(* Logix 5000 project; controller PBS_Perfusion vendor 1 type 14 code 217 rev 32.14; software revision 32.03; part 12 of 27 *)
(* tags used below, declared in another part *)
   Inp_OvrdCmd : DINT;   // Override Device Command: 0=None, 1=St.0, 2=St.1, 3=St.2, 4=St.3
   Cfg_NumStates : DINT;   // Number of device states (2..4)
   Cfg_OutSt0Write : SINT;   // Bit=1: write output in state 0, Bit=0: leave in last state
   Cfg_OutSt0State : SINT;   // (if written) Bit=1: output set in State 0, Bit=0: output cleared
   Cfg_OutSt1Write : SINT;   // Bit=1: write output in state 1, Bit=0: leave in last state
   Cfg_OutSt1State : SINT;   // (if written) Bit=1: output set in State 1, Bit=0: output cleared
   Cfg_OutSt2Write : SINT;   // Bit=1: write output in state 2, Bit=0: leave in last state
   Cfg_OutSt2State : SINT;   // (if written) Bit=1: output set in State 2, Bit=0: output cleared
   Cfg_OutSt3Write : SINT;   // Bit=1: write output in state 3, Bit=0: leave in last state
   Cfg_OutSt3State : SINT;   // (if written) Bit=1: output set in State 3, Bit=0: output cleared
   Cfg_FdbkSt0Check : SINT;   // Bit=1: Check Feedback in state 0, Bit=0: don't care
   Cfg_FdbkSt1Check : SINT;   // Bit=1: Check Feedback in state 1, Bit=0: don't care
   Cfg_FdbkSt2Check : SINT;   // Bit=1: Check Feedback in state 2, Bit=0: don't care
   Cfg_FdbkSt3Check : SINT;   // Bit=1: Check Feedback in state 3, Bit=0: don't care
   Cfg_OperSt0Prio : BOOL;   // 1=OCmd_St0 any time, 0=OCmd_St0 only when Oper selected
   Cfg_OCmdResets : BOOL;   // 1=New device OCmd resets shed latches and cleared alarms, 0=OCmdReset req'd.
   PSet_Owner : DINT;   // Program Owner Request ID (non-zero) or Release (zero)
   PCmd_St0 : BOOL;   // Program Command to set device to State 0
   PCmd_St1 : BOOL;   // Program Command to set device to State 1
   PCmd_St2 : BOOL;   // Program Command to set device to State 2
   PCmd_St3 : BOOL;   // Program Command to set device to State 3
   XCmd_St0 : BOOL;   // External Command to set device to State 0
   XCmd_St1 : BOOL;   // External Command to set device to State 1
   XCmd_St2 : BOOL;   // External Command to set device to State 2
   XCmd_St3 : BOOL;   // External Command to set device to State 3
   Out_A : BOOL;   // Output A to Device
   Out_B : BOOL;   // Output B to Device
   Out_C : BOOL;   // Output C to Device
   Out_D : BOOL;   // Output D to Device
   Out_Horn : BOOL;   // 1=Sound audible prior to commanded energize/ state change
   Val_Cmd : DINT;   // Device Command 0=None, 1=State 0, 2=State 1, 3=State 2, 4=State 3
   Val_Owner : DINT;   // Current Object Owner ID (0=not owned)
   Sts_St0 : BOOL;   // 1=Device commanded to and confirmed in State 0
   Sts_St1 : BOOL;   // 1=Device commanded to and confirmed in State 1
   Sts_St2 : BOOL;   // 1=Device commanded to and confirmed in State 2
   Sts_St3 : BOOL;   // 1=Device commanded to and confirmed in State 3
   Sts_Moving : BOOL;   // 1=Device not yet confirmed in commended state
   Sts_Horn : BOOL;   // 1=Sound audible prior to commanded energize/ state change
   Sts_NotRdy : BOOL;   // 1=Device Not Ready, see detail bits for reason
   Nrdy_CfgErr : BOOL;   // 1=Device Not Ready: Configuration Error
   Nrdy_EqpFault : BOOL;   // 1=Device Not Ready: External Equipment Fault (Fault or Shed Requires Reset)
   Nrdy_Fail : BOOL;   // 1=Device Not Ready: Device Failure (Shed Requires Reset)
   Nrdy_IOFault : BOOL;   // 1=Device Not Ready: I/O Fault (Shed Requires Reset)
   Nrdy_PrioSt0 : BOOL;   // 1=Device Not Ready: Oper/Ext Priority State 0 Command Requires Reset
   Nrdy_Perm : BOOL;   // 1=Device Not Ready: Permissive Not OK
   Sts_OoS : ALIAS FOR CmdSrc.Sts_OoS;
   Sts_Maint : ALIAS FOR CmdSrc.Sts_Maint;
   Sts_Oper : ALIAS FOR CmdSrc.Sts_Oper;
   Sts_DeviceFault : ALIAS FOR DeviceFault.Inp;   // 1=Device Fault (from Inp_DeviceFault)
   P_D4SD : BOOL;   // Unique Parameter Name for auto - discovery
   Wrk_OutDPulseT : TIMER;   // Output D Pulse Timer
   Wrk_OutCPulseT : TIMER;   // Output C Pulse Timer
   Wrk_OutBPulseT : TIMER;   // Output B Pulse Timer
   Wrk_OutAPulseT : TIMER;   // Output A Pulse Timer
   Wrk_ActState : DINT;   // Actual State (enum)
   Fail : P_Alarm;   // Device Fail to reach commanded position
   DeviceFault : P_Alarm;   // Device Fault from device via input
   CmdSrc : P_CmdSrc;   // Control / Command Source Selection
   IntlkTrip : P_Alarm;   // Interlock Trip Alarm
   Wrk_Out : SINT;   // Outputs (buffered) as a SINT for byte-wise operations
   Wrk_PermOK3 : BOOL;   // 1=Permissives are OK to go to state 3
   Wrk_PermOK2 : BOOL;   // 1=Permissives are OK to go to state 2
   Wrk_PermOK1 : BOOL;   // 1=Permissives are OK to go to state 1
   Wrk_PermOK0 : BOOL;   // 1=Permissives are OK to go to state 0
   Wrk_TgtState : DINT;   // Target device state as a number (0, 1, 2 or 3)
   Wrk_NewCmd : BOOL;   // 1=A state command has been received (even for same state)
   Wrk_PrevTgt : DINT;   // Previous Target State (last scan)
   Wrk_NotRdy : BOOL;   // Device Not Ready conditions excluding shed latches
   ORdy_St3 : BOOL;   // 1=Ready for OCmd_St3, enable HMI button
   ORdy_St2 : BOOL;   // 1=Ready for OCmd_St2, enable HMI button
   ORdy_St1 : BOOL;   // 1=Ready for OCmd_St1, enable HMI button
   ORdy_St0 : BOOL;   // 1=Ready for OCmd_St0, enable HMI button
   MRdy_Check : BOOL;   // 1=Ready for MCmd_Check, enable HMI button
   MRdy_Bypass : BOOL;   // 1=Ready for MCmd_Bypass, enable HMI button
   OCmd_St3 : BOOL;   // Operator Command to set device to State 3
   OCmd_St2 : BOOL;   // Operator Command to set device to State 2
   OCmd_St1 : BOOL;   // Operator Command to set device to State 1
   OCmd_St0 : BOOL;   // Operator Command to set device to State 0
   MCmd_Check : BOOL;   // Maintenance Command to Check Interlocks and Permissives
   MCmd_Bypass : BOOL;   // Maintenance Command to Bypass Interlocks and Permissives
   Wrk_StartHorn : BOOL;   // 1=Sound audible prior to commanded energize/ state change
   REAL : DINT;
(* P_D4SD, continued *)

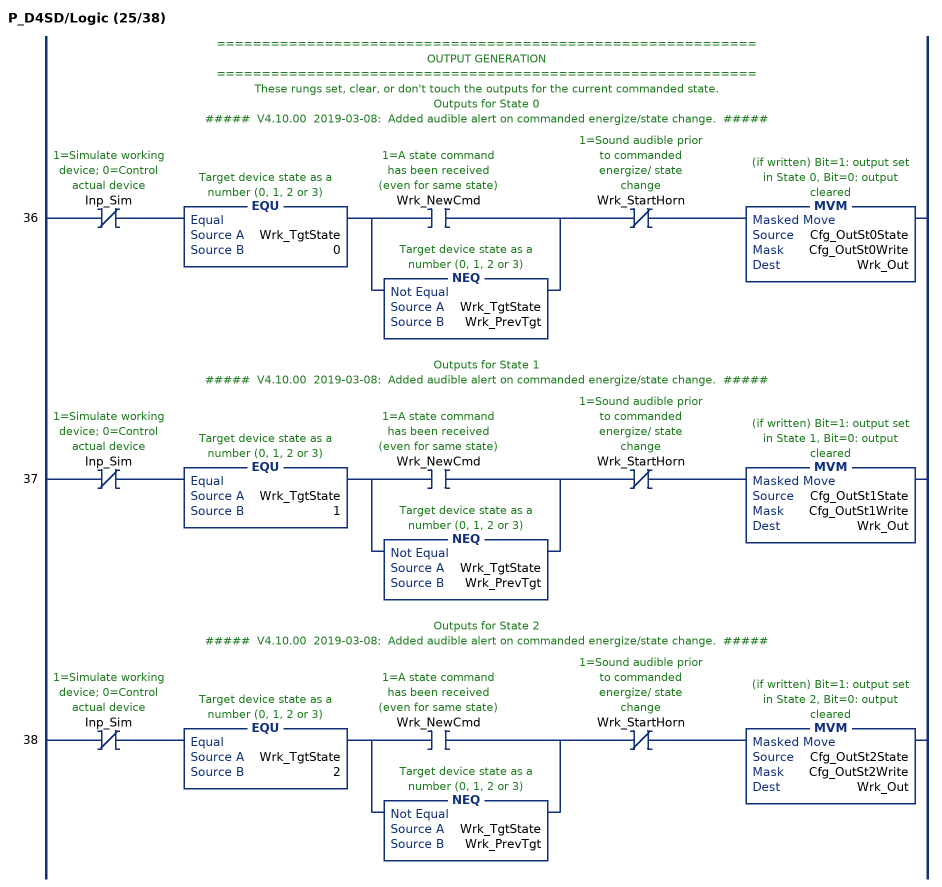
   // ============================================================
   // OUTPUT GENERATION
   // ============================================================
   // These rungs set, clear, or don't touch the outputs for the current commanded state.
   // Outputs for State 0
   // #####  V4.10.00  2019-03-08:  Added audible alert on commanded energize/state change.  #####
   36: XIO(Inp_Sim)EQU(Wrk_TgtState,0)[XIC(Wrk_NewCmd) ,NEQ(Wrk_TgtState,Wrk_PrevTgt) ]XIO(Wrk_StartHorn)MVM(Cfg_OutSt0State,Cfg_OutSt0Write,Wrk_Out);
   // Outputs for State 1
   // #####  V4.10.00  2019-03-08:  Added audible alert on commanded energize/state change.  #####
   37: XIO(Inp_Sim)EQU(Wrk_TgtState,1)[XIC(Wrk_NewCmd) ,NEQ(Wrk_TgtState,Wrk_PrevTgt) ]XIO(Wrk_StartHorn)MVM(Cfg_OutSt1State,Cfg_OutSt1Write,Wrk_Out);
   // Outputs for State 2
   // #####  V4.10.00  2019-03-08:  Added audible alert on commanded energize/state change.  #####
   38: XIO(Inp_Sim)EQU(Wrk_TgtState,2)[XIC(Wrk_NewCmd) ,NEQ(Wrk_TgtState,Wrk_PrevTgt) ]XIO(Wrk_StartHorn)MVM(Cfg_OutSt2State,Cfg_OutSt2Write,Wrk_Out);
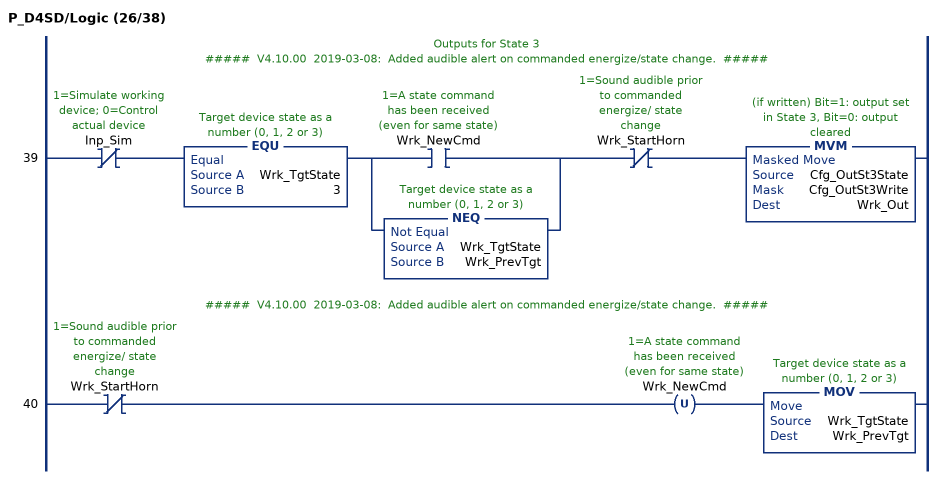
   // Outputs for State 3
   // #####  V4.10.00  2019-03-08:  Added audible alert on commanded energize/state change.  #####
   39: XIO(Inp_Sim)EQU(Wrk_TgtState,3)[XIC(Wrk_NewCmd) ,NEQ(Wrk_TgtState,Wrk_PrevTgt) ]XIO(Wrk_StartHorn)MVM(Cfg_OutSt3State,Cfg_OutSt3Write,Wrk_Out);
   // #####  V4.10.00  2019-03-08:  Added audible alert on commanded energize/state change.  #####
   40: XIO(Wrk_StartHorn)OTU(Wrk_NewCmd)MOV(Wrk_TgtState,Wrk_PrevTgt);
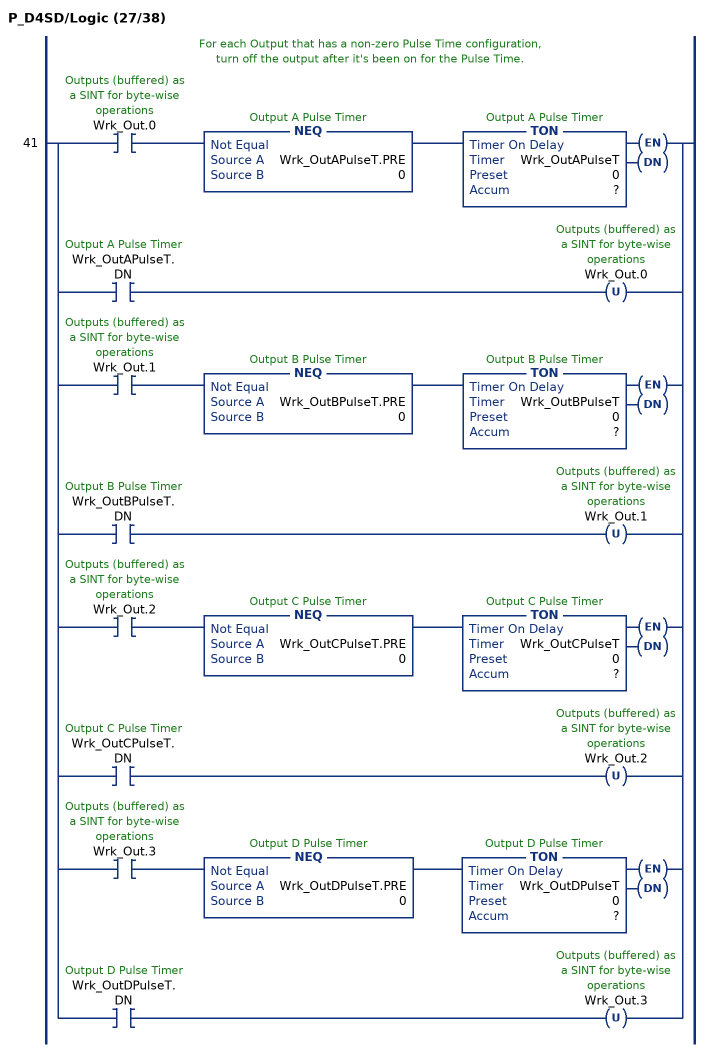
   // For each Output that has a non-zero Pulse Time configuration,
   // turn off the output after it's been on for the Pulse Time.
   41: [XIC(Wrk_Out.0) NEQ(Wrk_OutAPulseT.PRE,0) TON(Wrk_OutAPulseT,?,?) ,XIC(Wrk_OutAPulseT.DN) OTU(Wrk_Out.0) ,XIC(Wrk_Out.1) NEQ(Wrk_OutBPulseT.PRE,0) TON(Wrk_OutBPulseT,?,?) ,XIC(Wrk_OutBPulseT.DN) OTU(Wrk_Out.1) ,XIC(Wrk_Out.2) NEQ(Wrk_OutCPulseT.PRE,0) TON(Wrk_OutCPulseT,?,?) ,XIC(Wrk_OutCPulseT.DN) OTU(Wrk_Out.2) ,XIC(Wrk_Out.3) NEQ(Wrk_OutDPulseT.PRE,0) TON(Wrk_OutDPulseT,?,?) ,XIC(Wrk_OutDPulseT.DN) OTU(Wrk_Out.3) ];
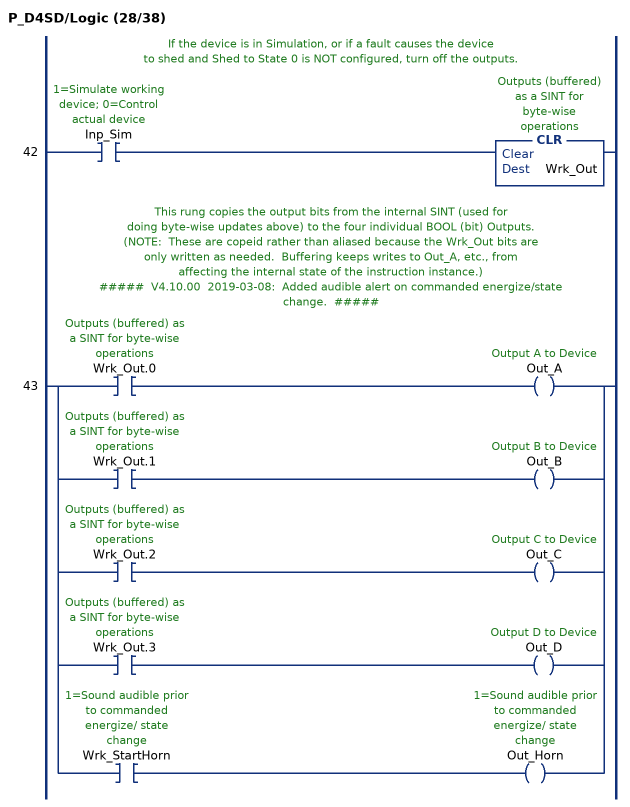
   // If the device is in Simulation, or if a fault causes the device
   // to shed and Shed to State 0 is NOT configured, turn off the outputs.
   42: XIC(Inp_Sim)CLR(Wrk_Out);
   // This rung copies the output bits from the internal SINT (used for
   // doing byte-wise updates above) to the four individual BOOL (bit) Outputs.
   // (NOTE:  These are copeid rather than aliased because the Wrk_Out bits are
   // only written as needed.  Buffering keeps writes to Out_A, etc., from
   // affecting the internal state of the instruction instance.)
   // #####  V4.10.00  2019-03-08:  Added audible alert on commanded energize/state change.  #####
   43: [XIC(Wrk_Out.0) OTE(Out_A) ,XIC(Wrk_Out.1) OTE(Out_B) ,XIC(Wrk_Out.2) OTE(Out_C) ,XIC(Wrk_Out.3) OTE(Out_D) ,XIC(Wrk_StartHorn) OTE(Out_Horn) ];
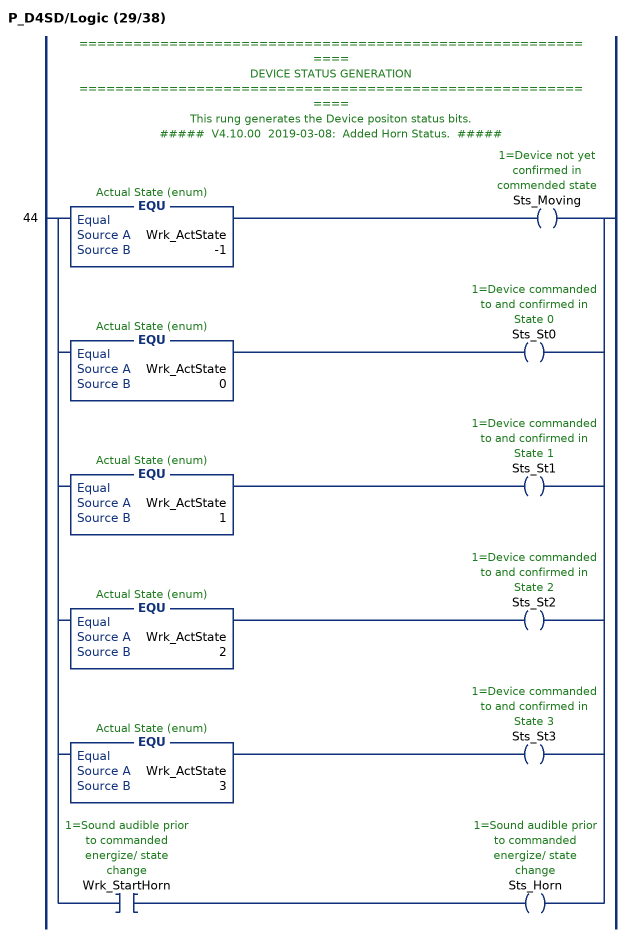
   // ============================================================
   // DEVICE STATUS GENERATION
   // ============================================================
   // This rung generates the Device positon status bits.
   // #####  V4.10.00  2019-03-08:  Added Horn Status.  #####
   44: [EQU(Wrk_ActState,-1) OTE(Sts_Moving) ,EQU(Wrk_ActState,0) OTE(Sts_St0) ,EQU(Wrk_ActState,1) OTE(Sts_St1) ,EQU(Wrk_ActState,2) OTE(Sts_St2) ,EQU(Wrk_ActState,3) OTE(Sts_St3) ,XIC(Wrk_StartHorn) OTE(Sts_Horn) ];
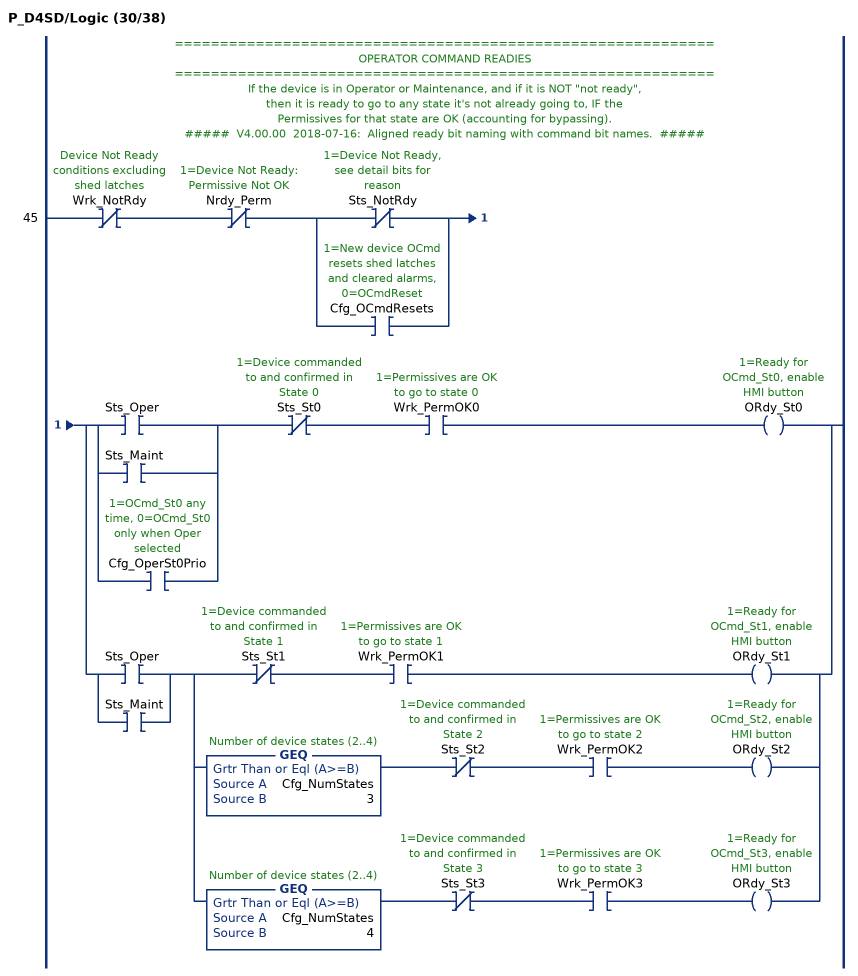
   // ============================================================
   // OPERATOR COMMAND READIES
   // ============================================================
   // If the device is in Operator or Maintenance, and if it is NOT "not ready",
   // then it is ready to go to any state it's not already going to, IF the
   // Permissives for that state are OK (accounting for bypassing).
   // #####  V4.00.00  2018-07-16:  Aligned ready bit naming with command bit names.  #####
   45: XIO(Wrk_NotRdy)XIO(Nrdy_Perm)[XIO(Sts_NotRdy) ,XIC(Cfg_OCmdResets) ][[XIC(Sts_Oper) ,XIC(Sts_Maint) ,XIC(Cfg_OperSt0Prio) ] XIO(Sts_St0) XIC(Wrk_PermOK0) OTE(ORdy_St0) ,[XIC(Sts_Oper) ,XIC(Sts_Maint) ] [XIO(Sts_St1) XIC(Wrk_PermOK1) OTE(ORdy_St1) ,GEQ(Cfg_NumStates,3) XIO(Sts_St2) XIC(Wrk_PermOK2) OTE(ORdy_St2) ,GEQ(Cfg_NumStates,4) XIO(Sts_St3) XIC(Wrk_PermOK3) OTE(ORdy_St3) ] ];
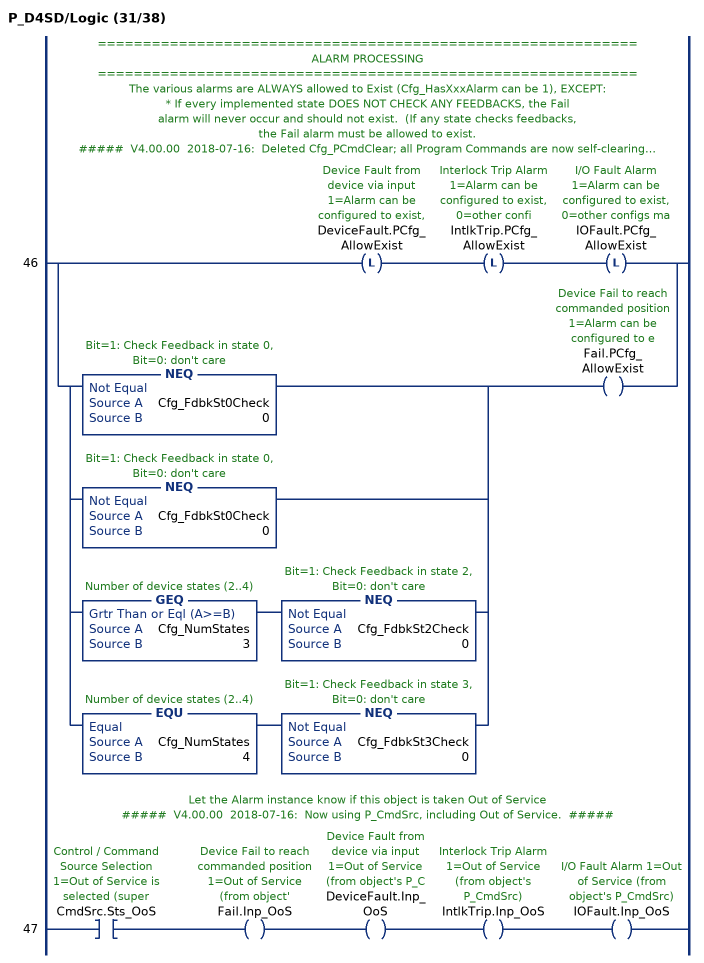
   // ============================================================
   // ALARM PROCESSING
   // ============================================================
   // The various alarms are ALWAYS allowed to Exist (Cfg_HasXxxAlarm can be 1), EXCEPT:
   // * If every implemented state DOES NOT CHECK ANY FEEDBACKS, the Fail
   // alarm will never occur and should not exist.  (If any state checks feedbacks,
   // the Fail alarm must be allowed to exist.
   // #####  V4.00.00  2018-07-16:  Deleted Cfg_PCmdClear; all Program Commands are now self-clearing.  #####
   46: [OTL(DeviceFault.PCfg_AllowExist) OTL(IntlkTrip.PCfg_AllowExist) OTL(IOFault.PCfg_AllowExist) ,[NEQ(Cfg_FdbkSt0Check,0) ,NEQ(Cfg_FdbkSt0Check,0) ,GEQ(Cfg_NumStates,3) NEQ(Cfg_FdbkSt2Check,0) ,EQU(Cfg_NumStates,4) NEQ(Cfg_FdbkSt3Check,0) ] OTE(Fail.PCfg_AllowExist) ];
   // Let the Alarm instance know if this object is taken Out of Service
   // #####  V4.00.00  2018-07-16:  Now using P_CmdSrc, including Out of Service.  #####
   47: XIC(CmdSrc.Sts_OoS)OTE(Fail.Inp_OoS)OTE(DeviceFault.Inp_OoS)OTE(IntlkTrip.Inp_OoS)OTE(IOFault.Inp_OoS);
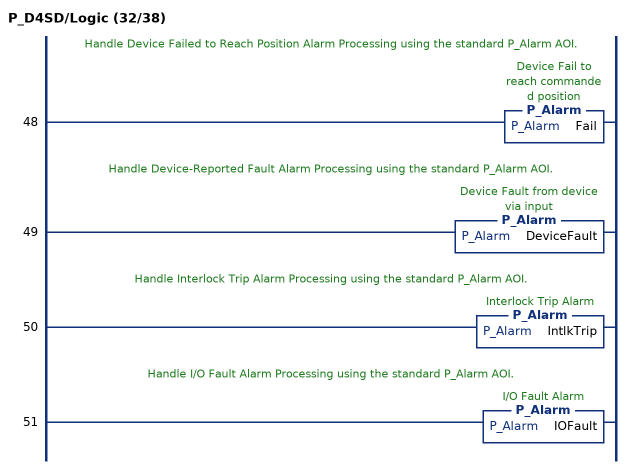
   // Handle Device Failed to Reach Position Alarm Processing using the standard P_Alarm AOI.
   48: P_Alarm(Fail);
   // Handle Device-Reported Fault Alarm Processing using the standard P_Alarm AOI.
   49: P_Alarm(DeviceFault);
   // Handle Interlock Trip Alarm Processing using the standard P_Alarm AOI.
   50: P_Alarm(IntlkTrip);
   // Handle I/O Fault Alarm Processing using the standard P_Alarm AOI.
   51: P_Alarm(IOFault);
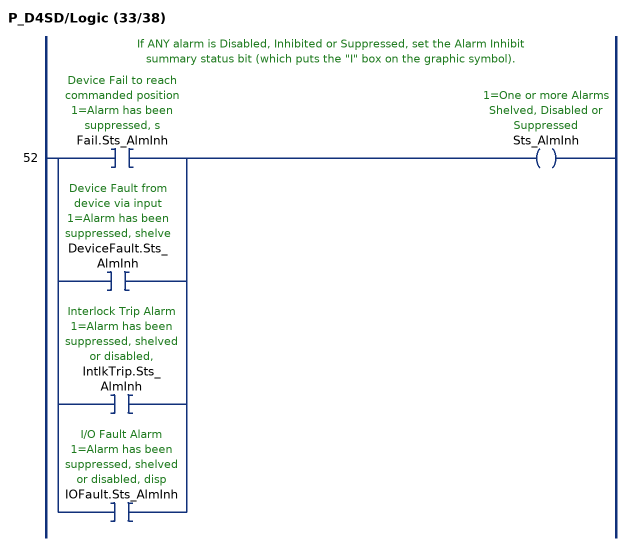
   // If ANY alarm is Disabled, Inhibited or Suppressed, set the Alarm Inhibit
   // summary status bit (which puts the "I" box on the graphic symbol).
   52: [XIC(Fail.Sts_AlmInh) ,XIC(DeviceFault.Sts_AlmInh) ,XIC(IntlkTrip.Sts_AlmInh) ,XIC(IOFault.Sts_AlmInh) ]OTE(Sts_AlmInh);
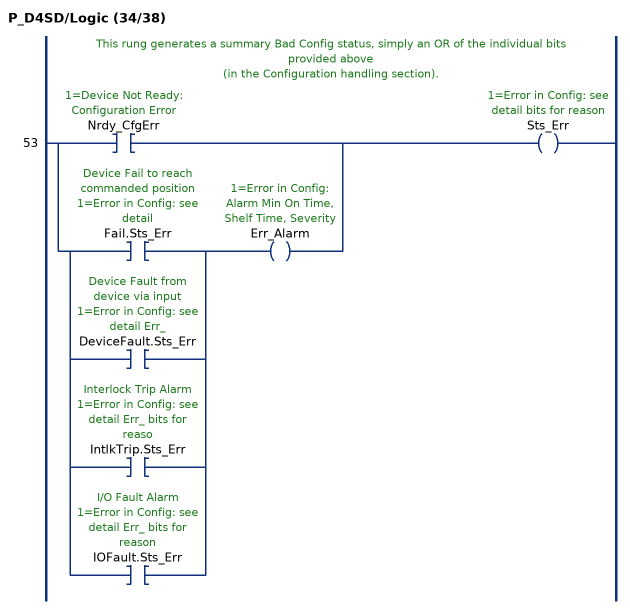
   // This rung generates a summary Bad Config status, simply an OR of the individual bits provided above
   // (in the Configuration handling section).
   53: [XIC(Nrdy_CfgErr) ,[XIC(Fail.Sts_Err) ,XIC(DeviceFault.Sts_Err) ,XIC(IntlkTrip.Sts_Err) ,XIC(IOFault.Sts_Err) ] OTE(Err_Alarm) ]OTE(Sts_Err);
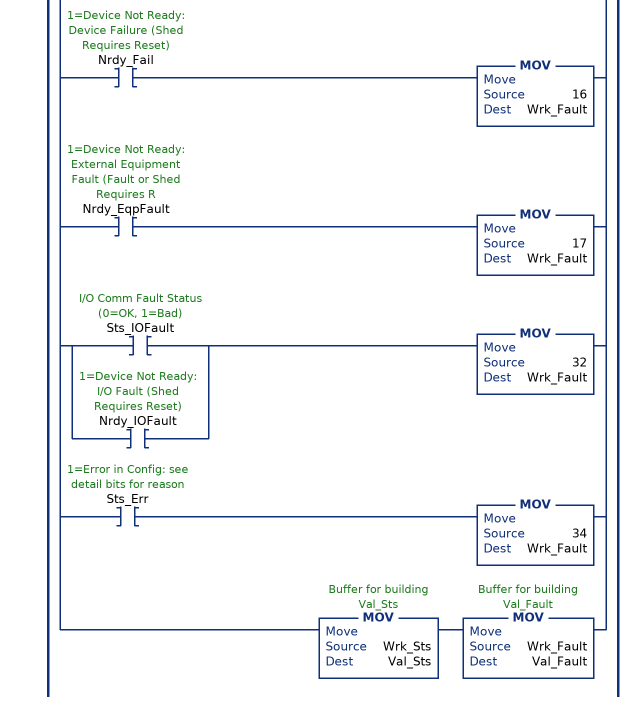
   // This rung generates the enumerated Device Status:
   // 0 = Powerup / Unknown
   // 1=Confirmed in State 0
   // 2 = Confirmed in State 1
   // 3 = Confirmed in State 2
   // 4 = Confirmed in State 3
   // 5 = Moving to new target State
   // 10 = Horn
   // And this rung generates the enumerated Device Fault Status:
   // 0 = none
   // 16 = Failed to reach commanded position
   // 17 = Device Fail (from input)
   // 32 = I/O Fault
   // 34 = Config Error
   // #####  V4.00.00  2018-07-16:  Disable/Enable replaced by P_CmdSrc Out of Service (OoS).  #####
   // #####  V4.10.00  2019-03-08:  Added Horn Status.  #####
   54: [CLR(Wrk_Sts) CLR(Wrk_Fault) ,XIC(Sts_St0) MOV(1,Wrk_Sts) ,XIC(Sts_St1) MOV(2,Wrk_Sts) ,XIC(Sts_St2) MOV(3,Wrk_Sts) ,XIC(Sts_St3) MOV(4,Wrk_Sts) ,XIC(Sts_Moving) MOV(9,Wrk_Sts) ,XIC(Sts_Horn) MOV(10,Wrk_Sts) ,XIC(Nrdy_Fail) MOV(16,Wrk_Fault) ,XIC(Nrdy_EqpFault) MOV(17,Wrk_Fault) ,[XIC(Sts_IOFault) ,XIC(Nrdy_IOFault) ] MOV(32,Wrk_Fault) ,XIC(Sts_Err) MOV(34,Wrk_Fault) ,MOV(Wrk_Sts,Val_Sts) MOV(Wrk_Fault,Val_Fault) ];
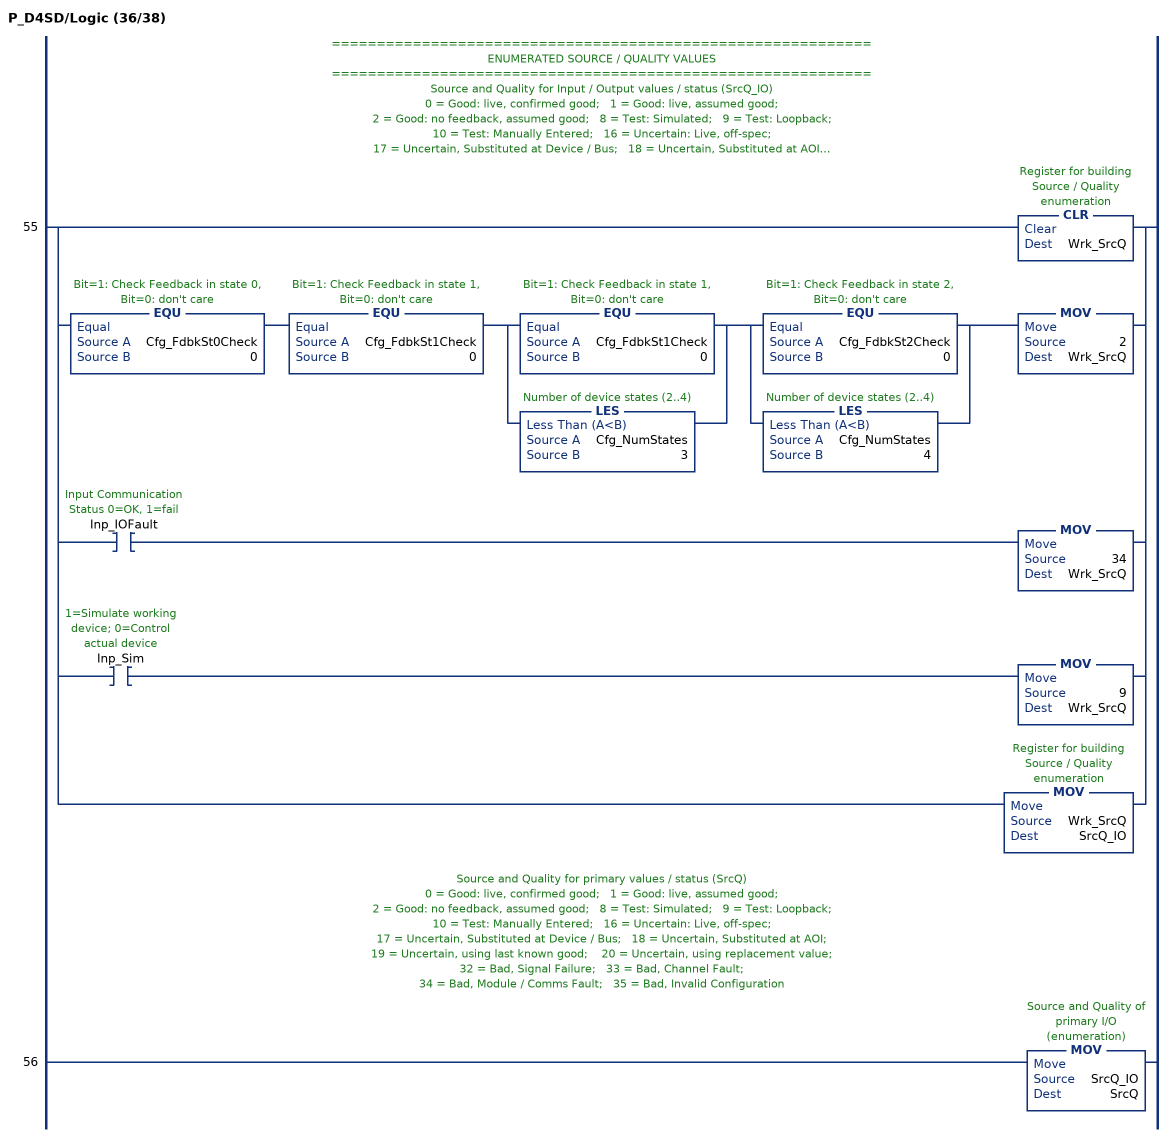
   // ============================================================
   // ENUMERATED SOURCE / QUALITY VALUES
   // ============================================================
   // Source and Quality for Input / Output values / status (SrcQ_IO)
   // 0 = Good: live, confirmed good;   1 = Good: live, assumed good;
   // 2 = Good: no feedback, assumed good;   8 = Test: Simulated;   9 = Test: Loopback;
   // 10 = Test: Manually Entered;   16 = Uncertain: Live, off-spec;
   // 17 = Uncertain, Substituted at Device / Bus;   18 = Uncertain, Substituted at AOI;
   // 19 = Uncertain, using last known good;    20 = Uncertain, using replacement value;
   // 32 = Bad, Signal Failure;   33 = Bad, Channel Fault;
   // 34 = Bad, Module / Comms Fault;   35 = Bad, Invalid Configuration.
   55: [CLR(Wrk_SrcQ) ,EQU(Cfg_FdbkSt0Check,0) EQU(Cfg_FdbkSt1Check,0) [EQU(Cfg_FdbkSt1Check,0) ,LES(Cfg_NumStates,3) ] [EQU(Cfg_FdbkSt2Check,0) ,LES(Cfg_NumStates,4) ] MOV(2,Wrk_SrcQ) ,XIC(Inp_IOFault) MOV(34,Wrk_SrcQ) ,XIC(Inp_Sim) MOV(9,Wrk_SrcQ) ,MOV(Wrk_SrcQ,SrcQ_IO) ];
   // Source and Quality for primary values / status (SrcQ)
   // 0 = Good: live, confirmed good;   1 = Good: live, assumed good;
   // 2 = Good: no feedback, assumed good;   8 = Test: Simulated;   9 = Test: Loopback;
   // 10 = Test: Manually Entered;   16 = Uncertain: Live, off-spec;
   // 17 = Uncertain, Substituted at Device / Bus;   18 = Uncertain, Substituted at AOI;
   // 19 = Uncertain, using last known good;    20 = Uncertain, using replacement value;
   // 32 = Bad, Signal Failure;   33 = Bad, Channel Fault;
   // 34 = Bad, Module / Comms Fault;   35 = Bad, Invalid Configuration
   56: MOV(SrcQ_IO,SrcQ);
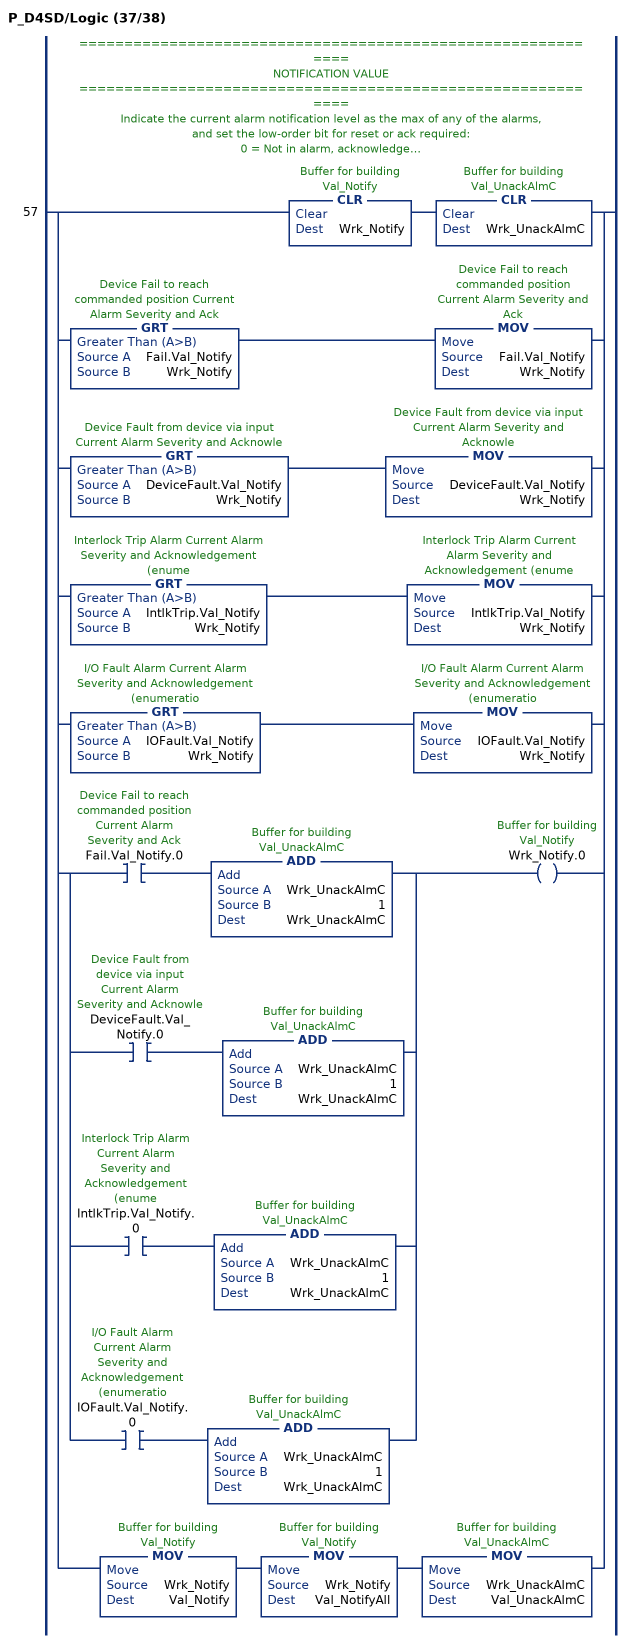
   // ============================================================
   // NOTIFICATION VALUE
   // ============================================================
   // Indicate the current alarm notification level as the max of any of the alarms,
   // and set the low-order bit for reset or ack required:
   // 0 = Not in alarm, acknowledged
   // 1 = Not in alarm, unacknowledged or reset required
   // 2 = Low severity alarm, acknowledged
   // 3 = Low severity alarm, unacknowledged
   // 4 = Medium severity alarm, acknowledged
   // 5 = Medium severity alarm, unacknowledged
   // 6 = High severity alarm, acknowledged
   // 7 = High severity alarm, unacknowledged
   // 8 = Urgent severity alarm, acknowledged
   // 9 = Urgent severity alarm, unacknowledged
   // #####  V4.00.00  2018-07-16:  Added Val_NotifyAll and Val_UnackAlmC to roll up alarm  #####
   // #####  priority / ack status and unack. alarm count.  #####
   57: [CLR(Wrk_Notify) CLR(Wrk_UnackAlmC) ,GRT(Fail.Val_Notify,Wrk_Notify) MOV(Fail.Val_Notify,Wrk_Notify) ,GRT(DeviceFault.Val_Notify,Wrk_Notify) MOV(DeviceFault.Val_Notify,Wrk_Notify) ,GRT(IntlkTrip.Val_Notify,Wrk_Notify) MOV(IntlkTrip.Val_Notify,Wrk_Notify) ,GRT(IOFault.Val_Notify,Wrk_Notify) MOV(IOFault.Val_Notify,Wrk_Notify) ,[XIC(Fail.Val_Notify.0) ADD(Wrk_UnackAlmC,1,Wrk_UnackAlmC) ,XIC(DeviceFault.Val_Notify.0) ADD(Wrk_UnackAlmC,1,Wrk_UnackAlmC) ,XIC(IntlkTrip.Val_Notify.0) ADD(Wrk_UnackAlmC,1,Wrk_UnackAlmC) ,XIC(IOFault.Val_Notify.0) ADD(Wrk_UnackAlmC,1,Wrk_UnackAlmC) ] OTE(Wrk_Notify.0) ,MOV(Wrk_Notify,Val_Notify) MOV(Wrk_Notify,Val_NotifyAll) MOV(Wrk_UnackAlmC,Val_UnackAlmC) ];
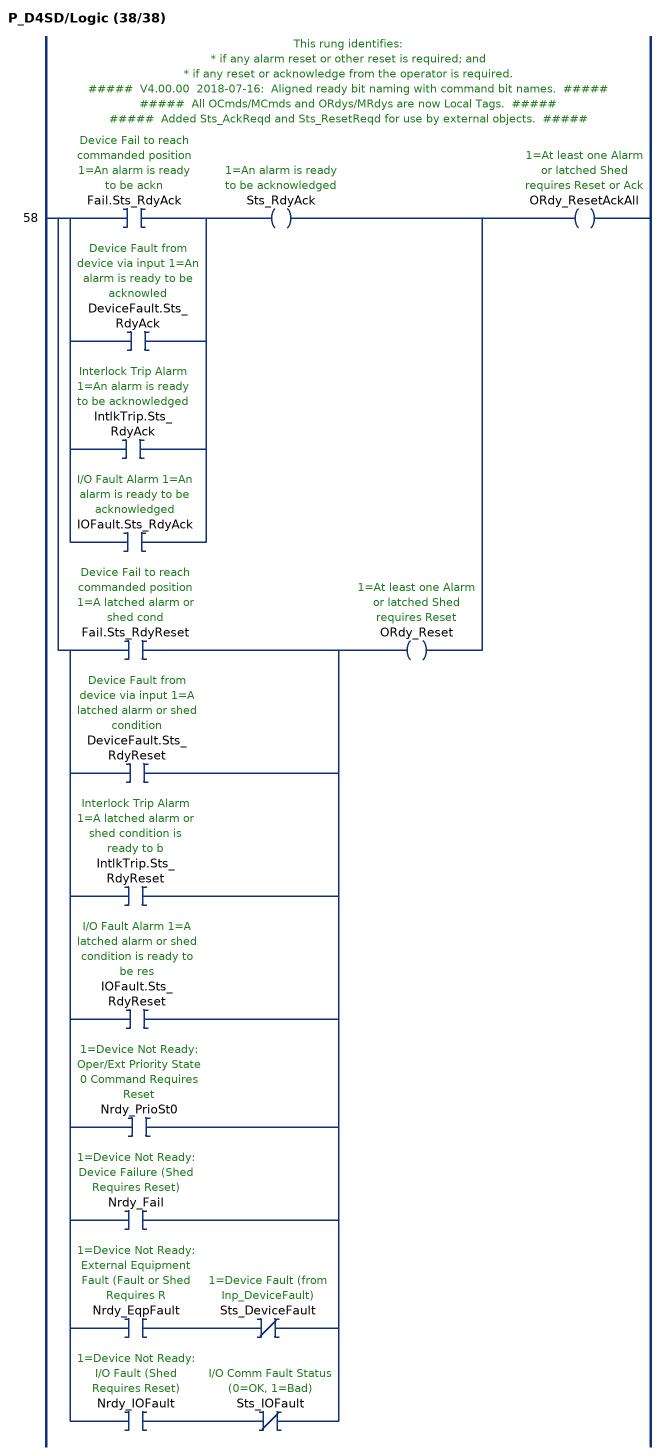
   // This rung identifies:
   // * if any alarm reset or other reset is required; and
   // * if any reset or acknowledge from the operator is required.
   // #####  V4.00.00  2018-07-16:  Aligned ready bit naming with command bit names.  #####
   // #####  All OCmds/MCmds and ORdys/MRdys are now Local Tags.  #####
   // #####  Added Sts_AckReqd and Sts_ResetReqd for use by external objects.  #####
   58: [[XIC(Fail.Sts_RdyAck) ,XIC(DeviceFault.Sts_RdyAck) ,XIC(IntlkTrip.Sts_RdyAck) ,XIC(IOFault.Sts_RdyAck) ] OTE(Sts_RdyAck) ,[XIC(Fail.Sts_RdyReset) ,XIC(DeviceFault.Sts_RdyReset) ,XIC(IntlkTrip.Sts_RdyReset) ,XIC(IOFault.Sts_RdyReset) ,XIC(Nrdy_PrioSt0) ,XIC(Nrdy_Fail) ,XIC(Nrdy_EqpFault) XIO(Sts_DeviceFault) ,XIC(Nrdy_IOFault) XIO(Sts_IOFault) ] OTE(ORdy_Reset) ]OTE(ORdy_ResetAckAll);
END_ROUTINE

ROUTINE Prescan   (* ladder *)
// Clear Ownership, clear "lurking" Commands
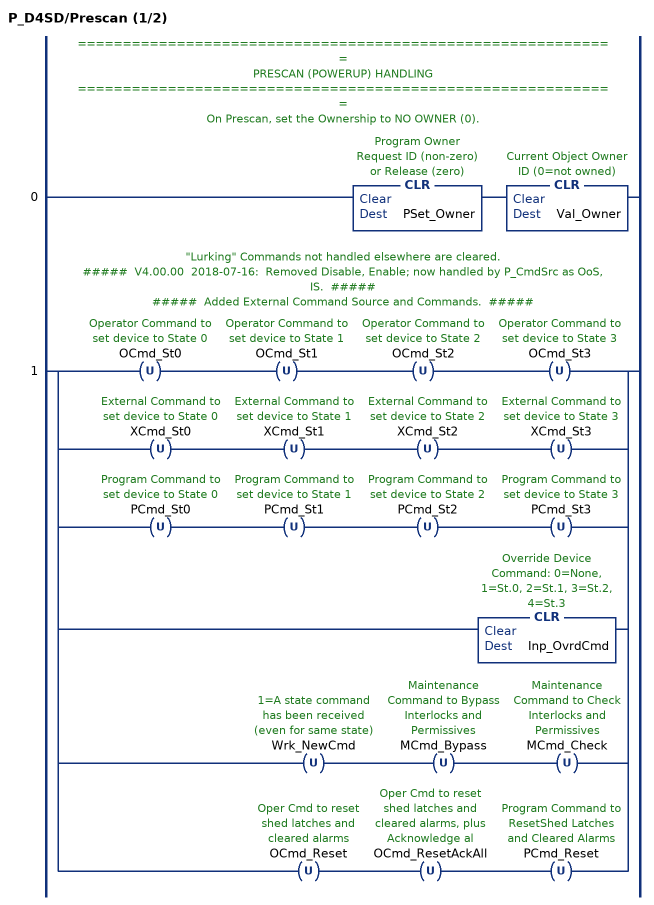
   // ============================================================
   // PRESCAN (POWERUP) HANDLING
   // ============================================================
   // On Prescan, set the Ownership to NO OWNER (0).
   0: CLR(PSet_Owner)CLR(Val_Owner);
   // "Lurking" Commands not handled elsewhere are cleared.
   // #####  V4.00.00  2018-07-16:  Removed Disable, Enable; now handled by P_CmdSrc as OoS, IS.  #####
   // #####  Added External Command Source and Commands.  #####
   1: [OTU(OCmd_St0) OTU(OCmd_St1) OTU(OCmd_St2) OTU(OCmd_St3) ,OTU(XCmd_St0) OTU(XCmd_St1) OTU(XCmd_St2) OTU(XCmd_St3) ,OTU(PCmd_St0) OTU(PCmd_St1) OTU(PCmd_St2) OTU(PCmd_St3) ,CLR(Inp_OvrdCmd) ,OTU(Wrk_NewCmd) OTU(MCmd_Bypass) OTU(MCmd_Check) ,OTU(OCmd_Reset) OTU(OCmd_ResetAckAll) OTU(PCmd_Reset) ];
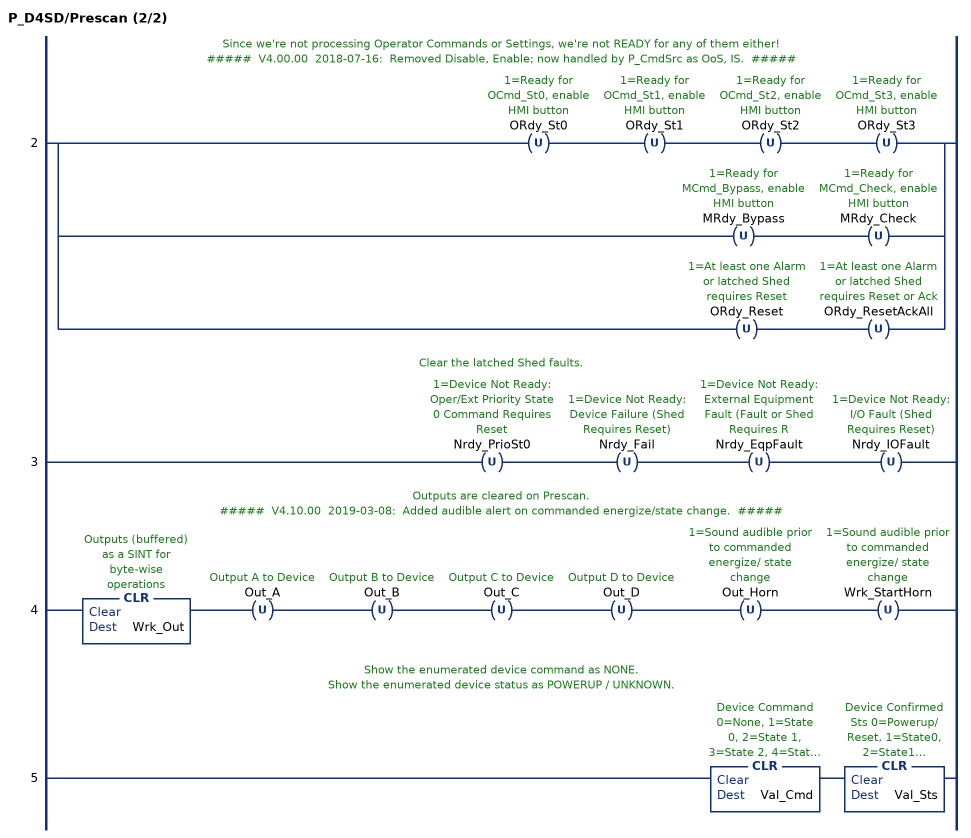
   // Since we're not processing Operator Commands or Settings, we're not READY for any of them either!
   // #####  V4.00.00  2018-07-16:  Removed Disable, Enable; now handled by P_CmdSrc as OoS, IS.  #####
   2: [OTU(ORdy_St0) OTU(ORdy_St1) OTU(ORdy_St2) OTU(ORdy_St3) ,OTU(MRdy_Bypass) OTU(MRdy_Check) ,OTU(ORdy_Reset) OTU(ORdy_ResetAckAll) ];
   // Clear the latched Shed faults.
   3: OTU(Nrdy_PrioSt0)OTU(Nrdy_Fail)OTU(Nrdy_EqpFault)OTU(Nrdy_IOFault);
   // Outputs are cleared on Prescan.
   // #####  V4.10.00  2019-03-08:  Added audible alert on commanded energize/state change.  #####
   4: CLR(Wrk_Out)OTU(Out_A)OTU(Out_B)OTU(Out_C)OTU(Out_D)OTU(Out_Horn)OTU(Wrk_StartHorn);
   // Show the enumerated device command as NONE.
   // Show the enumerated device status as POWERUP / UNKNOWN.
   5: CLR(Val_Cmd)CLR(Val_Sts);
END_ROUTINE
END_ADD_ON_INSTRUCTION

ADD_ON_INSTRUCTION P_DIn   (* revision 4.10 .00 Release, vendor Rockwell Automation, ExecutePrescan, ExecuteEnableInFalse *)
// Discrete Input
// Revision note:
// See Instruction Help for a summary of changes, and see 4.10 Release Notes for details.
// Help:
// Copyright © Rockwell Automation, Inc.  All Rights Reserved.
// This instruction monitors a discrete (1 / 0) input and checks for alarm conditions.
// The Inp_Gate input must be set (=1, its default value) and the alarm enabled for
// the Target Disagree alarm to occur.  This alarm will not occur until the Inp_Gate
// input has been set for the Gate Delay (Cfg_GateDly) time.  The Gate is used to
// enable the alarm when some other condition is true; for example, a high vibration
// switch should only generate a Target Disagree alarm when the associated motor
// has been running long enough to stabilize.
// The Target Disagree alarm is generated when the Inp_PV (process variable)
// input is different from the Inp_Target (target) input.  The Target indicates the
// "normal" condition.  For example, a flow switch should indicate flow when a
// pump is running and should not indicate flow when a pump is stopped.  The
// pump run status is used as the Target input, and when the switch does not
// match the target (within the allotted time), the Target Disagree Alarm (e.g.,
// Flow Switch Failure) is generated.
// NOTE: the Inp_PV is inverted when the rung condition is false -- this allows the
// input to be a condition on the rung with P_DIn rather than mapped into Inp_PV.
// See P_DIn reference manual for details.
// This instruction includes a substitute PV capability for a manually-entered state.
// This may be useful when a sensor is out for repair or for simulation and testing.
// Alarms are provided by P_Alarm AOI instances.
// Target Disagree Status gating provided by a P_Gate AOI instance.
// SUMMARY OF CHANGES FROM PREVIOUS VERSION (4.00.00)
// See 4.10 Release Notes for details.
// * Added Cfg_HasMoreObj.
// SUMMARY OF CHANGES FROM PREVIOUS VERSION (3.5-01)
// See 4.00 Release Notes for details.
// * Changed Inf_ items to HMI_, and added Cfg_Area for security.
// * Added notify and unack count rollup for Channel object.
// * Added I/O Fault alarm.
// * Deleted Cfg_PCmdClear.  All Program Commands are now self-clearing.
// * Aligned ready bit naming with command bit names.
// * All OCmds/MCmds and ORdys/MRdys are now Local Tags.
// * Added Sts_RdyAck and Sts_RdyReset for use by external objects.
// * Changed delay time configuration items to REAL seconds.
VAR_INPUT
   Inp_PV : BOOL := 1; {visible}   // Input Signal (process variable) from Sensor
   Inp_IOFault : BOOL; {visible}   // Input Comm Status or Quality 1=Bad, 0=OK
   Inp_PVNotify : DINT;   // Related PV object alarm prio and ack status (enum)
   Inp_Target : BOOL := 1; {visible}   // Target State of Input (Disagree Status if not in Target State)
   Inp_Gate : ALIAS FOR TgtDisagreeGate.Inp_Gate; {visible}   // Gate Condition (=1 to enable Disagree Status)
   Inp_Sim : BOOL;   // 1=Use simulated PV (Set_SimPV); 0=Use Input (Inp_PV)
   Inp_Reset : BOOL;   // 1=Reset Alarm requiring reset
   Cfg_NoSubstPV : BOOL;   // 1=Disallow selection of Substitute PV
   Cfg_NormTextVis : BOOL := 1;   // 1=Display state text in "normal" state (= target), 0=hide (some HMI objects)
   Cfg_HasMoreObj : BOOL;   // 1=Tells HMI an object with more info is available
   Cfg_HasTgtDisagreeAlm : ALIAS FOR TgtDisagree.Cfg_Exists;   // 1=Target Disagree Alarm exists and will be checked
   Cfg_TgtDisagreeResetReqd : ALIAS FOR TgtDisagree.Cfg_ResetReqd;   // 1=Target Disagree Alarm is latched in, requires Reset Command to clear
   Cfg_TgtDisagreeAckReqd : ALIAS FOR TgtDisagree.Cfg_AckReqd;   // 1=Target Disagree Alarm must be acknowledged
   Cfg_HasIOFaultAlm : ALIAS FOR IOFault.Cfg_Exists;   // 1=Target Disagree Alarm exists and will be checked
   Cfg_IOFaultResetReqd : ALIAS FOR IOFault.Cfg_ResetReqd;   // 1=Target Disagree Alarm is latched in, requires Reset Command to clear
   Cfg_IOFaultAckReqd : ALIAS FOR IOFault.Cfg_AckReqd;   // 1=Target Disagree Alarm must be acknowledged
   Cfg_TgtDisagreeSeverity : ALIAS FOR TgtDisagree.Cfg_Severity;   // Target Disagree Alarm Severity: 1..250=Low, 251..500=Medium, 501..750=High, 751..1000=Urgent
   Cfg_IOFaultSeverity : ALIAS FOR IOFault.Cfg_Severity;   // Target Disagree Alarm Severity: 1..250=Low, 251..500=Medium, 501..750=High, 751..1000=Urgent
   Cfg_Debounce : REAL;   // Minimum time Input Sts must maintain state (sec)
   Cfg_GateDly : ALIAS FOR TgtDisagreeGate.Cfg_GateDly;   // Time Inp_Gate must be true before Disagree Status is checked (sec)
   Cfg_TgtDisagreeOnDly : ALIAS FOR TgtDisagreeGate.Cfg_OnDly;   // Minimum time for Input to disagree with Target to raise Status (sec)
   Cfg_TgtDisagreeOffDly : ALIAS FOR TgtDisagreeGate.Cfg_OffDly;   // Minimum time for Input to agree with Target to clear Status (sec)
   Set_SimPV : BOOL;   // PV used in Simulation (Inp_Sim=1)
   PCmd_Reset : BOOL;   // Program Command to Reset all latched Alarms
   PCmd_TgtDisagreeAck : ALIAS FOR TgtDisagree.PCmd_Ack;   // Program Command to Acknowledge the Target Disagree Alarm
   PCmd_TgtDisagreeSuppress : ALIAS FOR TgtDisagree.PCmd_Suppress;   // Program Command to Suppress the Target Disagree Alarm
   PCmd_TgtDisagreeUnsuppress : ALIAS FOR TgtDisagree.PCmd_Unsuppress;   // Program Command to Unsuppress the Target Disagree Alarm
   PCmd_TgtDisagreeUnshelve : ALIAS FOR TgtDisagree.PCmd_Unshelve;   // Program Command to Unshelve the Target Disagree Alarm
   PCmd_IOFaultAck : ALIAS FOR IOFault.PCmd_Ack;   // Program Command to Acknowledge the I/O Fault Alarm
   PCmd_IOFaultSuppress : ALIAS FOR IOFault.PCmd_Suppress;   // Program Command to Suppress the I/O Fault Alarm
   PCmd_IOFaultUnsuppress : ALIAS FOR IOFault.PCmd_Unsuppress;   // Program Command to Unsuppress the I/O Fault Alarm
   PCmd_IOFaultUnshelve : ALIAS FOR IOFault.PCmd_Unshelve;   // Program Command to Unshelve the I/O Fault Alarm
END_VAR
VAR_OUTPUT
   SrcQ_IO : DINT; {access Read Only}   // Source and Quality of primary I/O (enumeration)
   SrcQ : DINT; {access Read Only}   // Source and Quality of primary Val/Sts (enumeration)
   Val_Sts : DINT; {access Read Only}   // Device Confirmed Sts 0=PV Good, 6=PV Bad, 7=Substitute PV
   Val_Fault : DINT; {access Read Only}   // Device Fault Status 0=none, 16=Tgt Disagree, 32=I/O comms., 34=CfgErr
   Val_NotifyAll : DINT; {access Read Only}   // Current Alarm Level and Acknowledgement (enumeration)
   Val_UnackAlmC : DINT; {access Read Only}   // Count of Unacknowledged Alarms
   Sts : BOOL; {access Read Only, visible}   // Discrete Input Status (incl. Debounce, Manual Override, if used)
   Sts_PV : BOOL; {access Read Only, visible}   // Discrete Input Status (actual, not subject to Override)
   Sts_SubstPV : BOOL; {access Read Only}   // 1=Using Substitute PV (Input being overridden)
   Sts_InpPV : BOOL; {access Read Only}   // 1=Using Input PV (normal)
   Sts_PVBad : BOOL; {access Read Only}   // Input Comm Status/ Quality (0=OK, 1=Bad)
   Sts_MaintByp : BOOL; {access Read Only}   // 1=Device has a Maintenance Bypass function active
   Sts_AlmInh : BOOL; {access Read Only}   // 1=One or more Alarms Shelved, Disabled or Suppressed
   Sts_Err : BOOL; {access Read Only, visible}   // 1=Error in Config: see detail bits for reason
   Err_Timer : BOOL; {access Read Only}   // 1=Error in Config: Invalid Timer Preset (use 0 to 2147483)
   Err_Alarm : BOOL; {access Read Only}   // 1=Error in Config: Alarm Min On Time, Shelf Time, Severity
   Sts_RdyReset : ALIAS FOR ORdy_Reset; {access Read Only}   // 1=A latched alarm or shed condition is ready to be reset
   Sts_RdyAck : BOOL; {access Read Only}   // 1=An alarm is ready to be acknowledged
   Sts_TgtDisagreeCmp : ALIAS FOR TgtDisagreeGate.Inp;   // Input vs. Target comparicon result 1=Disagree
   Sts_TgtDisagreeGate : ALIAS FOR TgtDisagreeGate.Sts_Gate; {access Read Only}   // Target Disagree Gate Delay Status, 1=done
   Sts_TgtDisagree : ALIAS FOR TgtDisagree.Inp;   // 1=Input is not in Target state
   Alm_TgtDisagree : ALIAS FOR TgtDisagree.Alm;   // 1=Alarm: Input is not in Target state
   Ack_TgtDisagree : ALIAS FOR TgtDisagree.Ack;   // 1=Target Disagree Alarm has been acknowledged
   Sts_TgtDisagreeDisabled : ALIAS FOR TgtDisagree.Disabled;   // 1=Target Disagree Alarm has been Disabled by Maintenance
   Sts_TgtDisagreeShelved : ALIAS FOR TgtDisagree.Shelved;   // 1=Target Disagree Alarm has been Shelved by Operator
   Sts_TgtDisagreeSuppressed : ALIAS FOR TgtDisagree.Suppressed;   // 1=Target Disagree Alarm has been Suppressed by Program
   Sts_IOFault : ALIAS FOR IOFault.Inp;   // 1=Input communication fault (Inp_IOFault = 1)
   Alm_IOFault : ALIAS FOR IOFault.Alm;   // 1=Alarm: Input communication fault
   Ack_IOFault : ALIAS FOR IOFault.Ack;   // 1=I/O Fault Alarm has been acknowledged
   Sts_IOFaultDisabled : ALIAS FOR IOFault.Disabled;   // 1=I/O Fault Alarm has been Disabled by Maintenance
   Sts_IOFaultShelved : ALIAS FOR IOFault.Shelved;   // 1=I/O Fault Alarm has been Shelved by Operator
   Sts_IOFaultSuppressed : ALIAS FOR IOFault.Suppressed;   // 1=I/O Fault Alarm has been Suppressed by Program
   P_DIn : BOOL;   // Unique Parameter Name for auto - discovery
END_VAR
VAR
   Cfg_Tag : STRING_20 := 'P_DIn';   // Tagname for display on HMI
   Cfg_Desc : STRING_40 := 'Discrete Input';   // Description for display on HMI
   Cfg_Label : STRING_20 := 'Discrete Input';   // Label for graphic symbol displayed on HMI
   Wrk_Status : BOOL; {access None}   // Internal Status (after Manual Override selection)
   TgtDisagree : P_Alarm := (Cfg_AckReqd := 1, Cfg_AllowShelve := 1, Cfg_AllowDisable := 1, Cfg_Severity := 750, Cfg_AlmMinOnT := 5, PCfg_AllowExist := 1, Ack := 1);   // Target Disagree Alarm
   Wrk_FallT : TIMER; {access None}   // Timer to ensure Status LOW time on falling edge
   Wrk_RiseT : TIMER; {access None}   // Timer to ensure Status HIGH time on rising edge
   Wrk_SubstPV : BOOL; {access None}   // Internal flag: Using Substitute PV
   Cfg_1StText : STRING_8 := 'On';   // Text to display in PV=1 State
   Cfg_0StText : STRING_8 := 'Off';   // Text to display in PV=0 State
   HMI_Tab : SINT;   // Tab to display (FTView ME)
   Wrk_Fault : DINT; {access None}   // Buffer for building Val_Fault
   Wrk_Sts : DINT; {access None}   // Buffer for building Val_Sts
   Wrk_SrcQ : DINT; {access None}   // Register for building Source / Quality enumeration
   HMI_Type : STRING_16 := 'P_DIn'; {access Read Only}   // Must contain AOI name, used for HMI and Information S/W
   TgtDisagreeGate : P_Gate := (Inp_Gate := 1);   // Target Disagree Condition Gate/Delay
   Val_Notify : DINT; {access Read Only}   // Highest Alarm prio and ack status this object only (enum)
   Wrk_Notify : DINT; {access None}   // Buffer for building Val_Notify
   Cfg_Area : STRING_Area := 'area01';   // Process Area for security
   HMI_Lib : STRING_12 := 'RA-BAS'; {access Read Only}   // Display Library for Faceplate call-up
   Wrk_UnackAlmC : DINT; {access None}   // Buffer for building Val_UnackAlmC
   IOFault : P_Alarm := (Cfg_AckReqd := 1, Cfg_AllowShelve := 1, Cfg_AllowDisable := 1, Cfg_Severity := 1000, Cfg_MaxShelfT := 480, Cfg_AlmMinOnT := 5, PCfg_AllowExist := 1, Ack := 1);   // I/O Fault Alarm
   OCmd_ResetAckAll : BOOL;   // Operator Command to Reset and Acknowledge all Alarms
   OCmd_Reset : BOOL;   // Operator Command to Reset all latched Alarms
   MCmd_InpPV : BOOL;   // Maintenance Command to use Input PV (normal)
   MCmd_SubstPV : BOOL;   // Maintenance Command to use Substitute PV (override input)
   ORdy_ResetAckAll : BOOL; {access Read Only}   // 1=Ready for OCmd_ResetAckAll (enables HMI button)
   ORdy_Reset : BOOL; {access Read Only}   // 1=Ready for OCmd_Reset (enables HMI button)
   MRdy_InpPV : BOOL; {access Read Only}   // 1=Ready for MCmd_InpPV (enables HMI button)
   MRdy_SubstPV : BOOL; {access Read Only}   // 1=Ready for MCmd_SubstPV (enables HMI button)
   MSet_SubstPV : BOOL;   // Maintenance-Entered Substitute PV
   Wrk_ErrDebounce : BOOL; {access None}   // Error in Debounce Timer configuration
END_VAR

ROUTINE EnableInFalse   (* ladder *)
// Same as main Logic routine, except Inp is inverted (for use in LD logic)
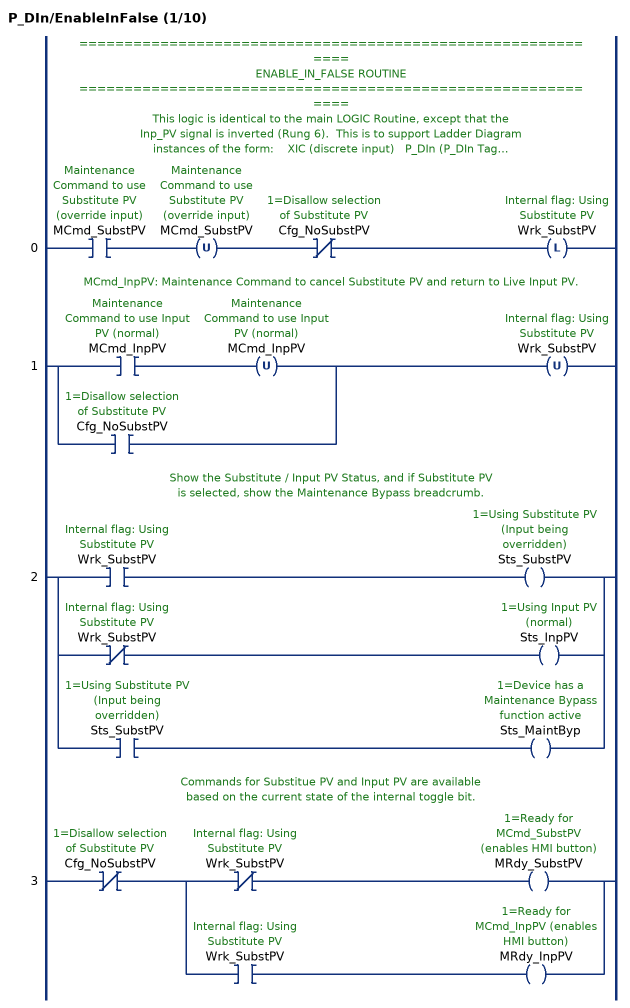
   // ============================================================
   // ENABLE_IN_FALSE ROUTINE
   // ============================================================
   // This logic is identical to the main LOGIC Routine, except that the
   // Inp_PV signal is inverted (Rung 6).  This is to support Ladder Diagram
   // instances of the form:    XIC (discrete input)   P_DIn (P_DIn Tag)
   // ============================================================
   // POWERUP / INVALID STATE HANDLING
   // ============================================================
   // All internal Work (state) bits maintain states through a power cycle and are
   // independent.  No Powerup / Invalid State Handling logic is required.
   // ============================================================
   // COMMAND PROCESSING
   // ============================================================
   // These rungs handle received Commands:
   // NOTE:  Operator Commands for P_Alarm are sent directly to the contained AOI.
   // MCmd_SubstPV: Maintenance Command to select Maintenance-entered substitute PV
   // Do not allow this Command if Cfg_NoSubstPV is set.
   0: XIC(MCmd_SubstPV)OTU(MCmd_SubstPV)XIO(Cfg_NoSubstPV)OTL(Wrk_SubstPV);
   // MCmd_InpPV: Maintenance Command to cancel Substitute PV and return to Live Input PV.
   1: [XIC(MCmd_InpPV) OTU(MCmd_InpPV) ,XIC(Cfg_NoSubstPV) ]OTU(Wrk_SubstPV);
   // Show the Substitute / Input PV Status, and if Substitute PV
   // is selected, show the Maintenance Bypass breadcrumb.
   2: [XIC(Wrk_SubstPV) OTE(Sts_SubstPV) ,XIO(Wrk_SubstPV) OTE(Sts_InpPV) ,XIC(Sts_SubstPV) OTE(Sts_MaintByp) ];
   // Commands for Substitue PV and Input PV are available
   // based on the current state of the internal toggle bit.
   3: XIO(Cfg_NoSubstPV)[XIO(Wrk_SubstPV) OTE(MRdy_SubstPV) ,XIC(Wrk_SubstPV) OTE(MRdy_InpPV) ];
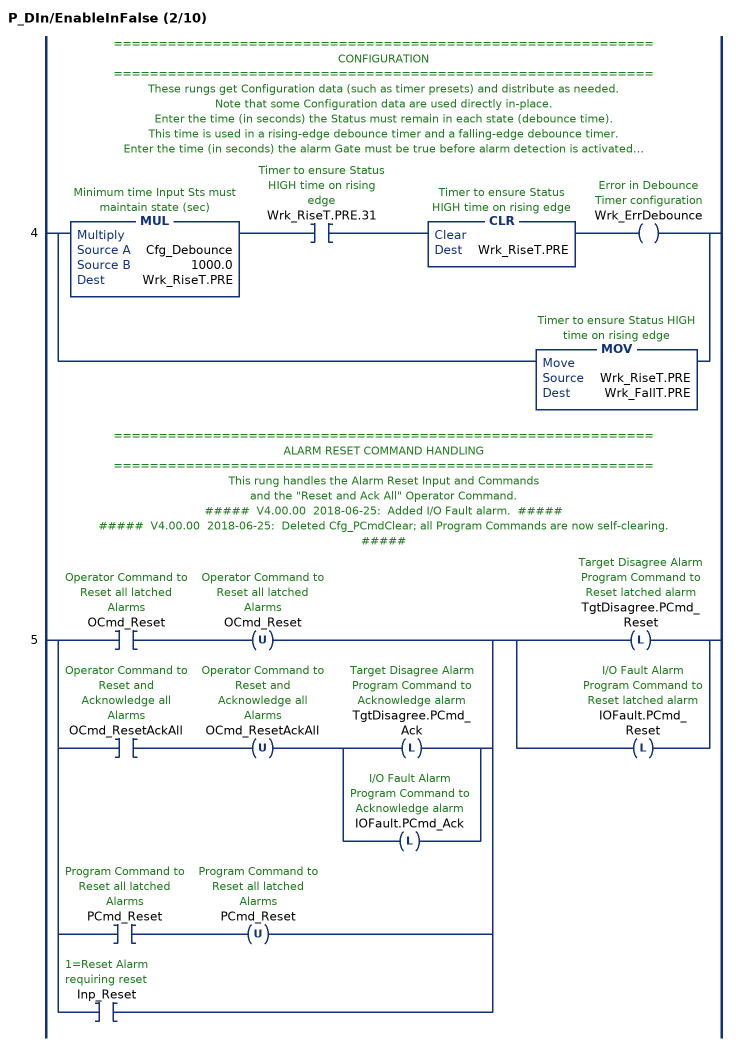
   // ============================================================
   // CONFIGURATION
   // ============================================================
   // These rungs get Configuration data (such as timer presets) and distribute as needed.
   // Note that some Configuration data are used directly in-place.
   // Enter the time (in seconds) the Status must remain in each state (debounce time).
   // This time is used in a rising-edge debounce timer and a falling-edge debounce timer.
   // Enter the time (in seconds) the alarm Gate must be true before alarm detection is activated.
   // Enter the On-Delay and Off-Delay times (in seconds) for the Target Disagree Status
   // (which feeds the Target Disagree Alarm).
   // If the timer preset calcuated wraps negative (more than 2.14... million seconds), then establish
   // a valid limit value for the Preset.  Note that a negative timer preset will fault the controller!!!
   // #####  V4.00.00  2018-06-25:  Changed delay time configuration items to REAL seconds.  #####
   4: [MUL(Cfg_Debounce,1000.0,Wrk_RiseT.PRE) XIC(Wrk_RiseT.PRE.31) CLR(Wrk_RiseT.PRE) OTE(Wrk_ErrDebounce) ,MOV(Wrk_RiseT.PRE,Wrk_FallT.PRE) ];
   // ============================================================
   // ALARM RESET COMMAND HANDLING
   // ============================================================
   // This rung handles the Alarm Reset Input and Commands
   // and the "Reset and Ack All" Operator Command.
   // #####  V4.00.00  2018-06-25:  Added I/O Fault alarm.  #####
   // #####  V4.00.00  2018-06-25:  Deleted Cfg_PCmdClear; all Program Commands are now self-clearing.  #####
   5: [XIC(OCmd_Reset) OTU(OCmd_Reset) ,XIC(OCmd_ResetAckAll) OTU(OCmd_ResetAckAll) [OTL(TgtDisagree.PCmd_Ack) ,OTL(IOFault.PCmd_Ack) ] ,XIC(PCmd_Reset) OTU(PCmd_Reset) ,XIC(Inp_Reset) ][OTL(TgtDisagree.PCmd_Reset) ,OTL(IOFault.PCmd_Reset) ];
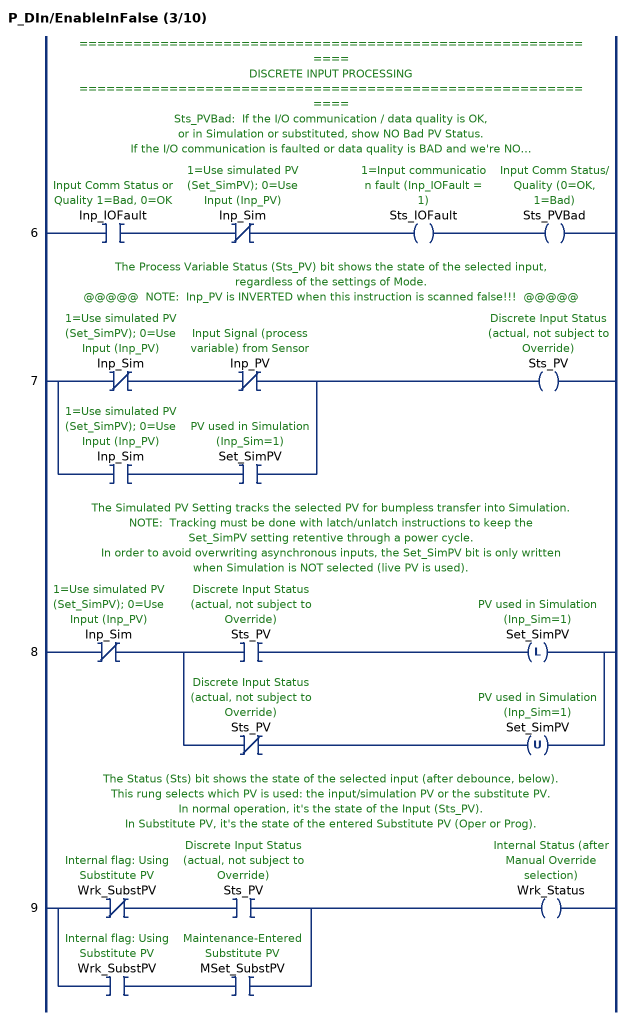
   // ============================================================
   // DISCRETE INPUT PROCESSING
   // ============================================================
   // Sts_PVBad:  If the I/O communication / data quality is OK,
   // or in Simulation or substituted, show NO Bad PV Status.
   // If the I/O communication is faulted or data quality is BAD and we're NOT
   // in Simulation or using substitute PV, show the Bad PV Status.
   // #####  V4.00.00  2018-06-25:  Added I/O Fault alarm.  #####
   6: XIC(Inp_IOFault)XIO(Inp_Sim)OTE(Sts_IOFault)OTE(Sts_PVBad);
   // The Process Variable Status (Sts_PV) bit shows the state of the selected input,
   // regardless of the settings of Mode.
   // @@@@@  NOTE:  Inp_PV is INVERTED when this instruction is scanned false!!!  @@@@@
   7: [XIO(Inp_Sim) XIO(Inp_PV) ,XIC(Inp_Sim) XIC(Set_SimPV) ]OTE(Sts_PV);
   // The Simulated PV Setting tracks the selected PV for bumpless transfer into Simulation.
   // NOTE:  Tracking must be done with latch/unlatch instructions to keep the
   // Set_SimPV setting retentive through a power cycle.
   // In order to avoid overwriting asynchronous inputs, the Set_SimPV bit is only written
   // when Simulation is NOT selected (live PV is used).
   8: XIO(Inp_Sim)[XIC(Sts_PV) OTL(Set_SimPV) ,XIO(Sts_PV) OTU(Set_SimPV) ];
   // The Status (Sts) bit shows the state of the selected input (after debounce, below).
   // This rung selects which PV is used: the input/simulation PV or the substitute PV.
   // In normal operation, it's the state of the Input (Sts_PV).
   // In Substitute PV, it's the state of the entered Substitute PV (Oper or Prog).
   9: [XIO(Wrk_SubstPV) XIC(Sts_PV) ,XIC(Wrk_SubstPV) XIC(MSet_SubstPV) ]OTE(Wrk_Status);
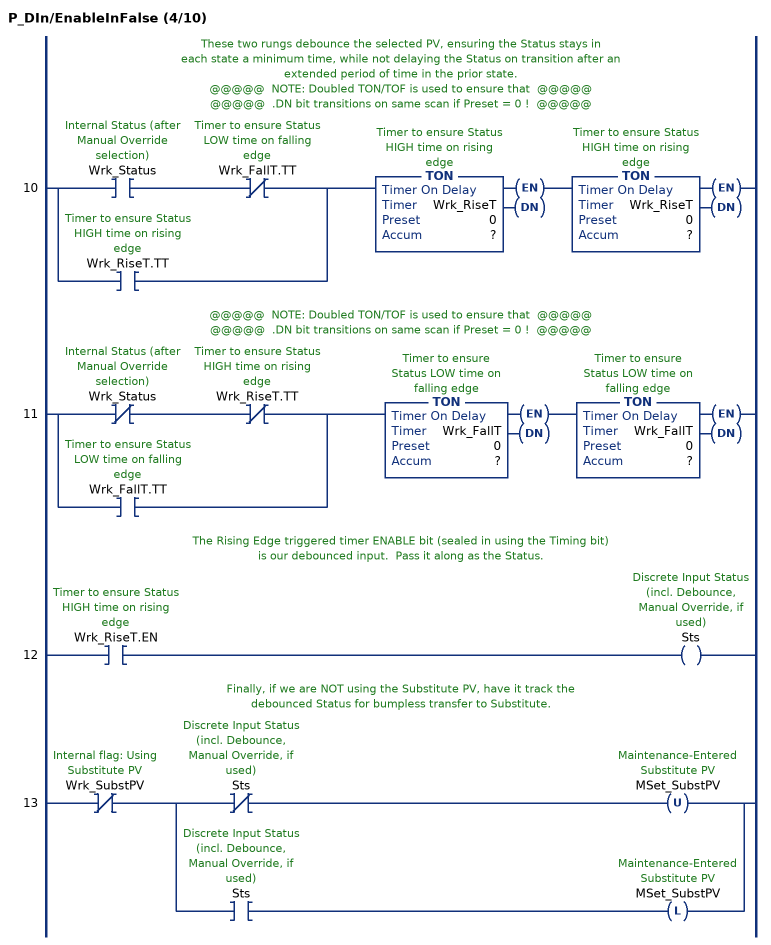
   // These two rungs debounce the selected PV, ensuring the Status stays in
   // each state a minimum time, while not delaying the Status on transition after an
   // extended period of time in the prior state.
   // @@@@@  NOTE: Doubled TON/TOF is used to ensure that  @@@@@
   // @@@@@  .DN bit transitions on same scan if Preset = 0 !  @@@@@
   10: [XIC(Wrk_Status) XIO(Wrk_FallT.TT) ,XIC(Wrk_RiseT.TT) ]TON(Wrk_RiseT,?,?)TON(Wrk_RiseT,?,?);
   // @@@@@  NOTE: Doubled TON/TOF is used to ensure that  @@@@@
   // @@@@@  .DN bit transitions on same scan if Preset = 0 !  @@@@@
   11: [XIO(Wrk_Status) XIO(Wrk_RiseT.TT) ,XIC(Wrk_FallT.TT) ]TON(Wrk_FallT,?,?)TON(Wrk_FallT,?,?);
   // The Rising Edge triggered timer ENABLE bit (sealed in using the Timing bit)
   // is our debounced input.  Pass it along as the Status.
   12: XIC(Wrk_RiseT.EN)OTE(Sts);
   // Finally, if we are NOT using the Substitute PV, have it track the
   // debounced Status for bumpless transfer to Substitute.
   13: XIO(Wrk_SubstPV)[XIO(Sts) OTU(MSet_SubstPV) ,XIC(Sts) OTL(MSet_SubstPV) ];
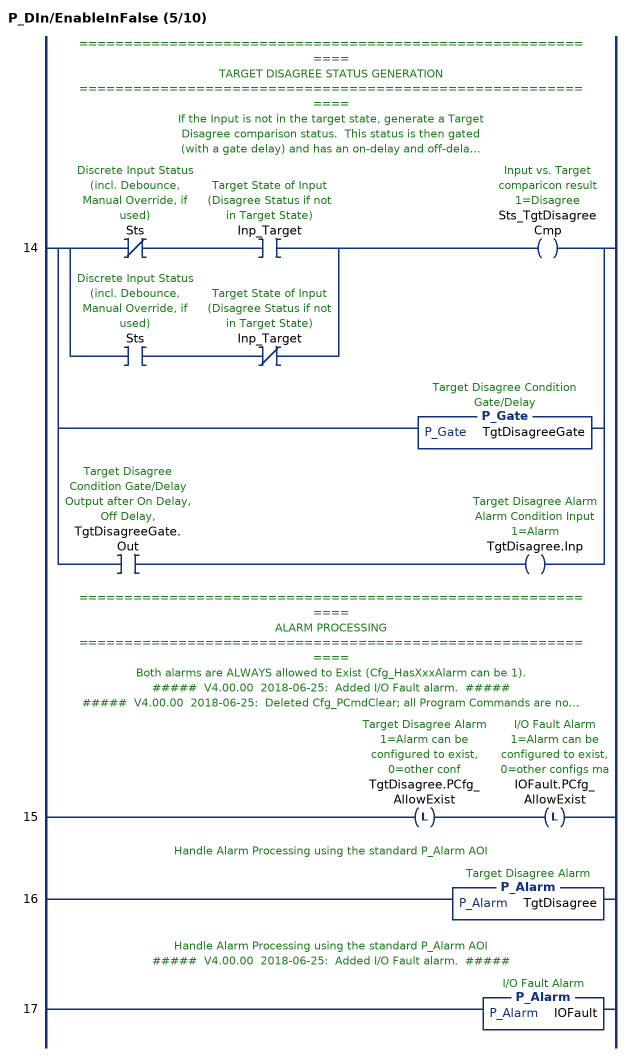
   // ============================================================
   // TARGET DISAGREE STATUS GENERATION
   // ============================================================
   // If the Input is not in the target state, generate a Target
   // Disagree comparison status.  This status is then gated
   // (with a gate delay) and has an on-delay and off-delay
   // before feeding the final Target Disagree status bit.
   14: [[XIO(Sts) XIC(Inp_Target) ,XIC(Sts) XIO(Inp_Target) ] OTE(Sts_TgtDisagreeCmp) ,P_Gate(TgtDisagreeGate) ,XIC(TgtDisagreeGate.Out) OTE(TgtDisagree.Inp) ];
   // ============================================================
   // ALARM PROCESSING
   // ============================================================
   // Both alarms are ALWAYS allowed to Exist (Cfg_HasXxxAlarm can be 1).
   // #####  V4.00.00  2018-06-25:  Added I/O Fault alarm.  #####
   // #####  V4.00.00  2018-06-25:  Deleted Cfg_PCmdClear; all Program Commands are now self-clearing.  #####
   15: OTL(TgtDisagree.PCfg_AllowExist)OTL(IOFault.PCfg_AllowExist);
   // Handle Alarm Processing using the standard P_Alarm AOI
   16: P_Alarm(TgtDisagree);
   // Handle Alarm Processing using the standard P_Alarm AOI
   // #####  V4.00.00  2018-06-25:  Added I/O Fault alarm.  #####
   17: P_Alarm(IOFault);
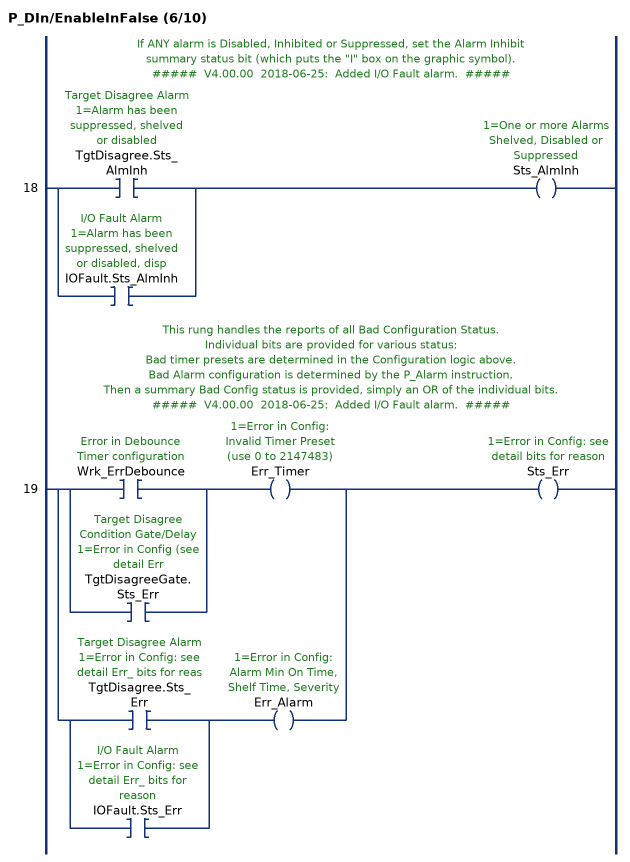
   // If ANY alarm is Disabled, Inhibited or Suppressed, set the Alarm Inhibit
   // summary status bit (which puts the "I" box on the graphic symbol).
   // #####  V4.00.00  2018-06-25:  Added I/O Fault alarm.  #####
   18: [XIC(TgtDisagree.Sts_AlmInh) ,XIC(IOFault.Sts_AlmInh) ]OTE(Sts_AlmInh);
   // This rung handles the reports of all Bad Configuration Status.
   // Individual bits are provided for various status:
   // Bad timer presets are determined in the Configuration logic above.
   // Bad Alarm configuration is determined by the P_Alarm instruction.
   // Then a summary Bad Config status is provided, simply an OR of the individual bits.
   // #####  V4.00.00  2018-06-25:  Added I/O Fault alarm.  #####
   19: [[XIC(Wrk_ErrDebounce) ,XIC(TgtDisagreeGate.Sts_Err) ] OTE(Err_Timer) ,[XIC(TgtDisagree.Sts_Err) ,XIC(IOFault.Sts_Err) ] OTE(Err_Alarm) ]OTE(Sts_Err);
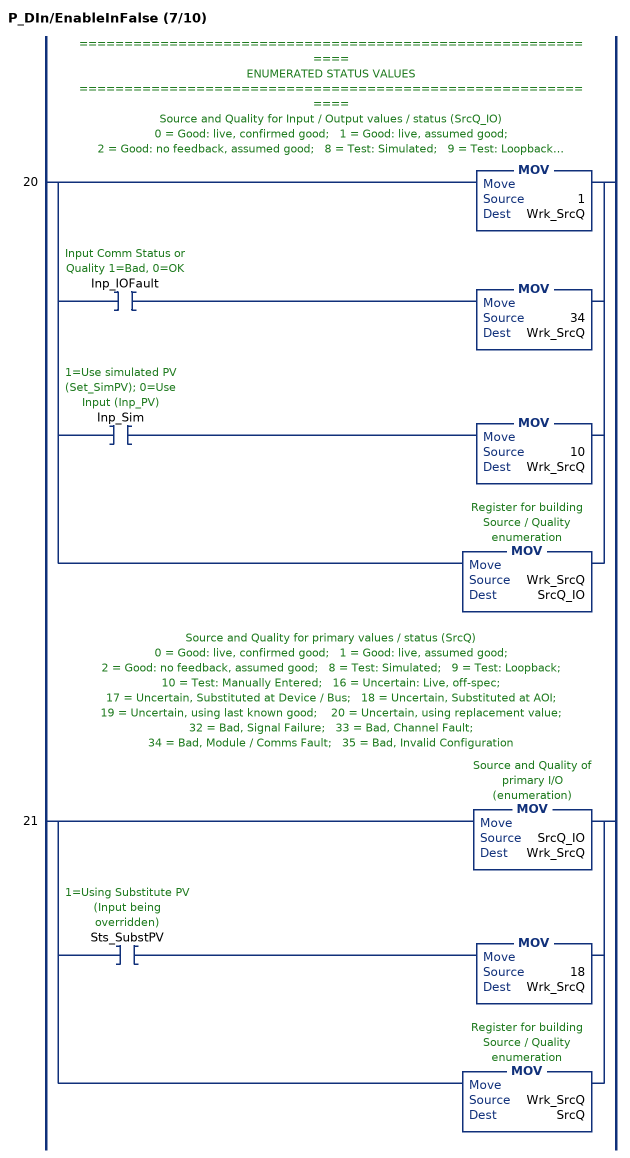
   // ============================================================
   // ENUMERATED STATUS VALUES
   // ============================================================
   // Source and Quality for Input / Output values / status (SrcQ_IO)
   // 0 = Good: live, confirmed good;   1 = Good: live, assumed good;
   // 2 = Good: no feedback, assumed good;   8 = Test: Simulated;   9 = Test: Loopback;
   // 10 = Test: Manually Entered;   16 = Uncertain: Live, off-spec;
   // 17 = Uncertain, Substituted at Device / Bus;   18 = Uncertain, Substituted at AOI;
   // 19 = Uncertain, using last known good;    20 = Uncertain, using replacement value;
   // 32 = Bad, Signal Failure;   33 = Bad, Channel Fault;
   // 34 = Bad, Module / Comms Fault;   35 = Bad, Invalid Configuration
   // #####  V4.00.00  2018-06-25:  Added I/O Fault alarm.  #####
   20: [MOV(1,Wrk_SrcQ) ,XIC(Inp_IOFault) MOV(34,Wrk_SrcQ) ,XIC(Inp_Sim) MOV(10,Wrk_SrcQ) ,MOV(Wrk_SrcQ,SrcQ_IO) ];
   // Source and Quality for primary values / status (SrcQ)
   // 0 = Good: live, confirmed good;   1 = Good: live, assumed good;
   // 2 = Good: no feedback, assumed good;   8 = Test: Simulated;   9 = Test: Loopback;
   // 10 = Test: Manually Entered;   16 = Uncertain: Live, off-spec;
   // 17 = Uncertain, Substituted at Device / Bus;   18 = Uncertain, Substituted at AOI;
   // 19 = Uncertain, using last known good;    20 = Uncertain, using replacement value;
   // 32 = Bad, Signal Failure;   33 = Bad, Channel Fault;
   // 34 = Bad, Module / Comms Fault;   35 = Bad, Invalid Configuration
   21: [MOV(SrcQ_IO,Wrk_SrcQ) ,XIC(Sts_SubstPV) MOV(18,Wrk_SrcQ) ,MOV(Wrk_SrcQ,SrcQ) ];
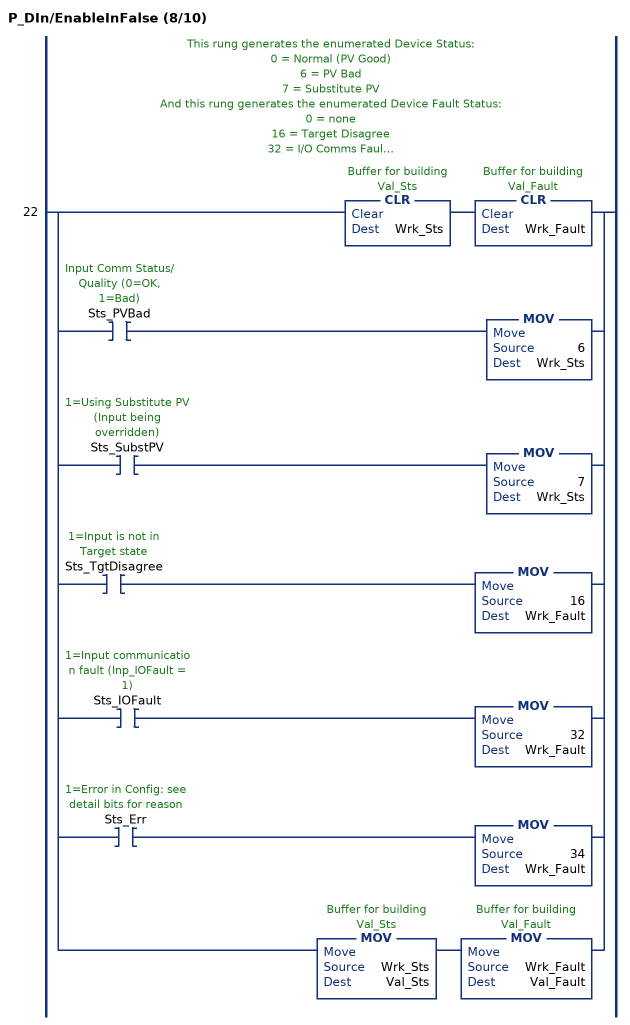
   // This rung generates the enumerated Device Status:
   // 0 = Normal (PV Good)
   // 6 = PV Bad
   // 7 = Substitute PV
   // And this rung generates the enumerated Device Fault Status:
   // 0 = none
   // 16 = Target Disagree
   // 32 = I/O Comms Fault
   // 34 = Config Error
   // #####  V4.00.00  2018-06-25:  Added I/O Fault alarm.  #####
   22: [CLR(Wrk_Sts) CLR(Wrk_Fault) ,XIC(Sts_PVBad) MOV(6,Wrk_Sts) ,XIC(Sts_SubstPV) MOV(7,Wrk_Sts) ,XIC(Sts_TgtDisagree) MOV(16,Wrk_Fault) ,XIC(Sts_IOFault) MOV(32,Wrk_Fault) ,XIC(Sts_Err) MOV(34,Wrk_Fault) ,MOV(Wrk_Sts,Val_Sts) MOV(Wrk_Fault,Val_Fault) ];
